ORGANIZATION_BLOCK "07_CYCL_FLT"
{ S7_Optimized_Access := 'FALSE' }
VERSION : 0.1
   VAR_TEMP
      OB80_EV_CLASS : Byte;
      OB80_FLT_ID : Byte;
      OB80_PRIORITY : Byte;
      OB80_OB_NUMBR : Byte;
      OB80_RESERVED_1 : Byte;
      OB80_RESERVED_2 : Byte;
      OB80_ERROR_INFO : Word;
      OB80_ERR_EV_CLASS : Byte;
      OB80_ERR_EV_NUM : Byte;
      OB80_OB_PRIORITY : Byte;
      OB80_OB_NUM : Byte;
      OB80_DATE_TIME : Date_And_Time;
   END_VAR


BEGIN
NETWORK
TITLE =


END_ORGANIZATION_BLOCK

